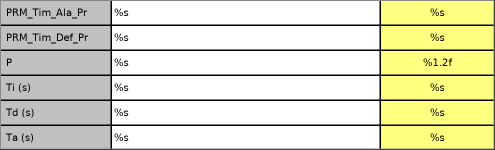
VISUALIZATION VISU_CONFIG_REGUL_GAZ  // 495x150
VAR_IN_OUT
	m_Input_REGULATION : BLOCK_REGUL_PR_GAZ;
END_VAR
    Rectangle (111,50 269x25), "%s", text list: 'TextList_Config_Gaz', text index: 31
    Rectangle (380,50 115x25), "%1.2f", text variable: m_Input_REGULATION.CONTROLEUR_GAZ.CONF_Kp, input disabled if: NOT Global_Variables.PRG_USER.ACTU_USER.CONF_MACHINE
        OnMouseDown: write the text variable via InputWithLimits, min 0
    Rectangle (0,50 111x25), "P", text variable: 1
    Rectangle (111,75 269x25), "%s", text list: 'TextList_Config_Gaz', text index: 32
    Rectangle (111,100 269x25), "%s", text list: 'TextList_Config_Gaz', text index: 33
    Rectangle (380,75 115x25), "%s", text variable: m_Input_REGULATION.CONTROLEUR_GAZ.CONF_Tn, input disabled if: NOT Global_Variables.PRG_USER.ACTU_USER.CONF_MACHINE
        OnMouseDown: write the text variable via InputWithLimits
    Rectangle (0,75 111x25), "Ti (s)", text variable: 1
    Rectangle (380,100 115x25), "%s", text variable: m_Input_REGULATION.CONTROLEUR_GAZ.CONF_Tv, input disabled if: NOT Global_Variables.PRG_USER.ACTU_USER.CONF_MACHINE
        OnMouseDown: write the text variable via InputWithLimits
    Rectangle (0,100 111x25), "Td (s)", text variable: 1
    Rectangle (111,125 269x25), "%s", text list: 'TextList_Config_Gaz', text index: 34
    Rectangle (380,125 115x25), "%s", text variable: m_Input_REGULATION.CONTROLEUR_GAZ.CONF_Td, input disabled if: NOT Global_Variables.PRG_USER.ACTU_USER.CONF_MACHINE
        OnMouseDown: write the text variable via InputWithLimits
    Rectangle (0,125 111x25), "Ta (s)", text variable: 1
    Rectangle (111,0 269x25), "%s", text list: 'TextList_Config_Gaz', text index: 29
    Rectangle (380,0 115x25), "%s", text variable: m_Input_REGULATION.PRM_Tim_Ala_Pr, input disabled if: NOT Global_Variables.PRG_USER.ACTU_USER.CONF_MACHINE
        OnMouseDown: write the text variable via InputWithLimits
    Rectangle (0,0 111x25), "PRM_Tim_Ala_Pr"
    Rectangle (111,25 269x25), "%s", text list: 'TextList_Config_Gaz', text index: 30
    Rectangle (380,25 115x25), "%s", text variable: m_Input_REGULATION.PRM_Tim_Def_Pr, input disabled if: NOT Global_Variables.PRG_USER.ACTU_USER.CONF_MACHINE
        OnMouseDown: write the text variable via InputWithLimits
    Rectangle (0,25 111x25), "PRM_Tim_Def_Pr"
END_VISUALIZATION

(* stored: Version 1.1.0.1, ProductVersion 3.1.4024.10
   Visu VISU_CONFIG_REGUL_GAZ: Id {ce4d0518-bb1b-418b-a1d0-37a4ff9c6cc2} *)
